(* Logix 5000 project; controller Capstone_PLC_1 1769-L16ER-BB1B rev 38.11; software revision 38.00 *)

TASK MainTask (continuous, watchdog 500 ms) : MainProgram, SecondaryProgram

MODULES
   Local : 1769-L16ER-BB1B (PointIO 0, rev 38.11)
      Point_IO : 1734-AENTR (Ethernet 192.168.1.30, rev 4.1, Output RPI 20 ms)   // Extended I/O for PLC
         POINT_DI_1 : 1734-IB8 (PointIO 1, rev 3.1)   // Sensors from tray to color identification
              Point_IO:1:I.2   // Induction sensor 2 - Extended I/O DI (1734-IB8, Slot 1, Channel 2)
              Point_IO:1:I.1   // Induction sensor 1 - Extended I/O DI (1734-IB8, Slot 1, Channel 1)
              Point_IO:1:I.0   // Tray present limit switch - Extended I/O DI (1734-IB8, Slot 1, Channel 0)
              Point_IO:1:I.3   // Induction sensor 3 - Extended I/O DI (1734-IB8, Slot 1, Channel 3)
              Point_IO:1:I.4   // Through beam sensor 1 - Extended I/O DI (1734-IB8, Slot 1, Channel 4)
              Point_IO:1:I.5   // Through beam sensor 2 - Extended I/O DI (1734-IB8, Slot 1, Channel 5)
         POINT_DI_2 : 1734-IB8 (PointIO 2, rev 3.1)   // Sorting sensors
              Point_IO:2:I.0   // Diffuse sensor, cube on conveyor - Extended I/O DI (1734-IB8, Slot 2, Channel 0)
              Point_IO:2:I.1   // Diffuse sensor, cube at bin 1 - Extended I/O DI (1734-IB8, Slot 2, Channel 1)
              Point_IO:2:I.2   // Diffuse sensor, cube at bin 2 - Extended I/O DI (1734-IB8, Slot 2, Channel 2)
              Point_IO:2:I.3   // Diffuse sensor, cube at bin 3 - Extended I/O DI (1734-IB8, Slot 2, Channel 3)
              Point_IO:2:I.4   // Diffuse sensor, cube at reject bin - Extended I/O DI (1734-IB8, Slot 2, Channel 4)
              Point_IO:2:I.5   // Input for color sensor bit 0
              Point_IO:2:I.6   // Input for color sensor bit 1
              Point_IO:2:I.7   // Input for color sensor bit 2
         POINT_DO_3 : 1734-OB8E (PointIO 3, rev 3.1)   // Conveyor, eject nozzles
              Point_IO:3:O.0   // Output for conveyor - Extended I/O DO (1734-OB8E, Slot 3, Channel 0)
              Point_IO:3:O.1   // Output for eject nozzle 1- Extended I/O DO (1734-OB8E, Slot 3, Channel 1)
              Point_IO:3:O.2   // Output for eject nozzle 2- Extended I/O DO (1734-OB8E, Slot 3, Channel 2)
              Point_IO:3:O.3   // Output for eject nozzle 3- Extended I/O DO (1734-OB8E, Slot 3, Channel 3)
      Discrete_IO : Embedded (PointIO 1, rev 38.1, Output RPI 20 ms)
END_MODULES

VAR_GLOBAL   (* controller tags *)
   At_Destination : BOOL;   // Tracks if the sorted cube has reached the correct bin
   Cmd_Conv : ALIAS FOR Point_IO:3:O.0;   // Logically commands conveyor output
   Cmd_Eject_1 : ALIAS FOR Point_IO:3:O.1;   // Logically commands ejection nozzle 1 output
   Cmd_Eject_2 : ALIAS FOR Point_IO:3:O.2;   // Logically commands ejection nozzle 2 output
   Cmd_Eject_3 : ALIAS FOR Point_IO:3:O.3;   // Logically commands ejection nozzle 3 output
   COL_DET : DINT := 4;   // State, detecting color
   Color_Bit_0 : ALIAS FOR Point_IO:2:I.5;   // Input from color sensor configured in Binary Out
   Color_Bit_1 : ALIAS FOR Point_IO:2:I.6;   // Input from color sensor configured in Binary Out
   Color_Bit_2 : ALIAS FOR Point_IO:2:I.7;   // Input from color sensor configured in Binary Out
   Color_Captured : BOOL;   // Triggers when a color has been identified successfully
   Color_Code : DINT;   // Detected color code
   ColorValid : BOOL;   // Validates color reading
   Con_0 : DINT;   // Constant 0
   Con_1 : DINT := 1;   // Constant 1
   Con_2 : DINT := 2;   // Constant 2
   Con_3 : DINT := 3;   // Constant 3
   Con_4 : DINT := 4;   // Constant 4
   Conv_Active : BOOL;   // Controls conveyor
   Count_1 : DINT;   // Bin 1 counter
   Count_2 : DINT;   // Bin 2 counter
   Count_3 : DINT;   // Bin 3 counter
   Count_4 : DINT;   // Bin 4 counter
   Dest_Bin : DINT;   // Stores destination bin after a cube is identified
   Destination_Known : BOOL;
   Detected_Color : DINT;   // Stores detected color code
   Dif_Bin_1 : ALIAS FOR Point_IO:2:I.1;   // Diffuse sensor: Bin 1
   Dif_Bin_2 : ALIAS FOR Point_IO:2:I.2;   // Diffuse sensor: Bin 2
   Dif_Bin_3 : ALIAS FOR Point_IO:2:I.3;   // Diffuse sensor: Bin 3
   Dif_Conv : ALIAS FOR Point_IO:2:I.0;   // Part detected on conveyor start position
   DONE : DINT := 7;   // State, cube sorted, triggers check, if cubes left to be sorted State returns to PICK, if not State returns to IDLE
   E_Stop : BOOL;   // Emergency stop, disables all outputs
   Eject_1 : BOOL;   // Controls ejection nozzle at bin 1
   Eject_2 : BOOL;   // Controls ejection nozzle at bin 2
   Eject_3 : BOOL;   // Controls ejection nozzle at bin 3
   FAULT : DINT := 99;
   HMI_Init_Sys : BOOL;   // HMI Input: Triggers SPEL_Init
   HMI_PB1 : ALIAS FOR STOP;   // HMI RED PB
   HMI_PB2 : BOOL;   // HMI ORANGE PB
   HMI_PB3 : ALIAS FOR START;   // HMI GREEN PB
   HMI_PB4 : BOOL;   // HMI BLUE PB
   HMI_Reset : BOOL;   // HMI Input to reset sysm to idle state
   IDLE : DINT := 1;   // State, system is initialized but no tray is present or tray present with no cubes
   Ind_Tray_1 : ALIAS FOR Point_IO:1:I.1;   // Induction sensor 1: Tray identification
   Ind_Tray_2 : ALIAS FOR Point_IO:1:I.2;   // Induction sensor 2: Tray identification
   Ind_Tray_3 : ALIAS FOR Point_IO:1:I.3;   // Induction sensor 3: Tray identification
   INIT : DINT;   // State, waiting for initialization conditions
   Lim_Tray_Pres : ALIAS FOR Point_IO:1:I.0;   // Limit switch: Tray presence
   OS_Col_Det : BOOL;   // Ensures color detetion only happens once on subroutine entry
   OS_Col_Det_State : BOOL;   // One shot ensures Col_Det state triggers cleanly
   OS_ColorValid : BOOL;   // Prevents multiple color readings at the same time
   OS_Conv : BOOL;   // One shot ensure clean transition to conveyor state
   OS_Init : BOOL;   // One shot keeps init executing once
   OS_Ready : BOOL;   // One shot protects IDLE > READY state transition
   OS_Reset : BOOL;   // One shot for reset to prevent it from triggering multiple times on a single press
   OS_Sort : BOOL;   // One shot ensure clean transition to sort state
   OS_Sort_Done : BOOL;   // One shot ensure clean entry into done state
   OS_Start : BOOL;   // One shot protects start production from triggering multiple times on input
   OS_TrayID_1 : BOOL;   // Protects from induction sensor reading multipletimes
   OS_TrayID_2 : BOOL;   // Protects from induction sensor reading multipletimes
   OS_TrayID_3 : BOOL;   // Protects from induction sensor reading multipletimes
   Output_Enable : BOOL;   // Enables outputs if robot initialized, system in run mode, and no faults or estop
   PB1 : ALIAS FOR Local:1:I.Data.0;   // RED PB
   PB2 : ALIAS FOR Local:1:I.Data.1;   // ORANGE PB
   PB3 : ALIAS FOR Local:1:I.Data.2;   // GREEN PB
   PB4 : ALIAS FOR Local:1:I.Data.3;   // BLUE PB
   PICK : DINT := 3;   // State, robot picking
   Pick_Done : BOOL;   // Triggers when SPEL pick is completed
   Pick_Index : DINT;   // Tracks cubes on tray for picking
   PL1 : ALIAS FOR Local:1:O.Data.0;   // RED LIGHT
   PL2 : ALIAS FOR Local:1:O.Data.1;   // ORANGE LIGHT
   PL3 : ALIAS FOR Local:1:O.Data.2;   // GREEN LIGHT
   PL4 : ALIAS FOR Local:1:O.Data.3;   // BLUE LIGHT
   PLACE_AOI : BOOL;
   Place_Done : BOOL;
   READY : DINT := 2;   // State, Tray and cubes present
   Rec_Color_Bin_1 : DINT;   // HMI input: color assigned to bin 1
   Rec_Color_Bin_2 : DINT;   // HMI input: color assigned to bin 2
   Rec_Color_Bin_3 : DINT;   // HMI input: color assigned to bin 3
   Rec_Color_Bin_4 : DINT;   // HMI input: color assigned to bin 4 "reject"
   ROBOT_BUSY : BOOL;
   ROBOT_DONE : BOOL;
   ROBOT_INIT : BOOL;
   Robot_Initialized : BOOL;   // Checks if robot is ready for production
   ROBOT_PICK_1 : BOOL;
   ROBOT_PICK_2 : BOOL;
   ROBOT_PICK_3 : BOOL;
   ROBOT_PICK_4 : BOOL;
   ROBOT_READY : BOOL;
   SCADA_Color : DINT;   // SCADA tag shows identified color
   SCADA_Conv : BOOL;   // SCADA tag shows conveyor activity
   SCADA_Count_1 : DINT;   // SCADA tag shows counter for bin 1
   SCADA_Count_2 : DINT;   // SCADA tag shows counter for bin 2
   SCADA_Count_3 : DINT;   // SCADA tag shows counter for bin 3
   SCADA_Count_4 : DINT;   // SCADA tag shows counter for bin 4
   SCADA_Dest : DINT;   // SCADA tag shows destination bin
   SCADA_State : DINT;   // SCADA tag shows current system state
   SCADA_TrayID : DINT;   // SCADA tag shows Tray ID
   SORT : DINT := 6;   // State, cube on conveyor
   Sort_Done : BOOL;   // Tracks if sorting is done
   SPEL_Init : BOOL;   // Triggers SPEL_Init AOI
   SPEL_Init_Done : BOOL;   // Checks if SPEL_Init is completed
   START : BOOL;   // Start production, triggered by PB3 (green) or HMI input
   State : DINT;   // Tracks system state for control flow
   STOP : BOOL;   // Stops production, triggered by PB1 (red) or HMI input
   Sys_Fault : BOOL;   // Enabled for any fault condition
   Sys_Rdy : BOOL;   // System staged and safe for production
   Sys_Run : BOOL;   // Production active
   TEST_Color_Entry : BOOL;   // User controlled bit for entering color detation, used for testing/debugging
   Thr_Cubes_1 : ALIAS FOR Point_IO:1:I.4;   // Through beam sensor: identifies cube presence in tray row 1
   Thr_Cubes_2 : ALIAS FOR Point_IO:1:I.5;   // Through beam sensor: identifies cube presence in tray row 2
   TIMER_BLINK_1 : TIMER := (PRE := 500);
   TIMER_BLINK_2 : TIMER := (PRE := 500);
   TIMER_EJECT_1 : TIMER := (PRE := 200);
   TIMER_EJECT_2 : TIMER := (PRE := 200);
   TIMER_EJECT_3 : TIMER := (PRE := 200);
   TIMER_REJECT : TIMER := (PRE := 8000);
   TMR_Color_Read : TIMER := (PRE := 500);   // Delays color sensor input for validation
   TO_CONV : DINT := 5;   // State, moving cube to conveyor
   Tray_Full : BOOL;   // Energizes if both through beam sensors are triggered for cube presence
   TrayID : DINT;   // Calculated tray ID from induction sensors
   TrayIdentified : BOOL;   // Tracks if a tray is identified
END_VAR

PROGRAM MainProgram   (* main routine MainRoutine *)

ROUTINE Blinker_Fault   (* ladder *)
// Flashes red light to indicate system fault
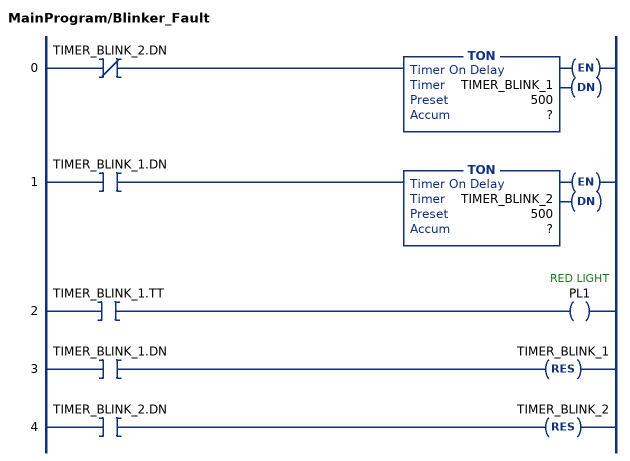
   0: XIO(TIMER_BLINK_2.DN)TON(TIMER_BLINK_1,?,?);
   1: XIC(TIMER_BLINK_1.DN)TON(TIMER_BLINK_2,?,?);
   2: XIC(TIMER_BLINK_1.TT)OTE(PL1);
   3: XIC(TIMER_BLINK_1.DN)RES(TIMER_BLINK_1);
   4: XIC(TIMER_BLINK_2.DN)RES(TIMER_BLINK_2);
END_ROUTINE

ROUTINE Blinker_Init   (* ladder *)
// Flashes blue light to show system ready for initialization
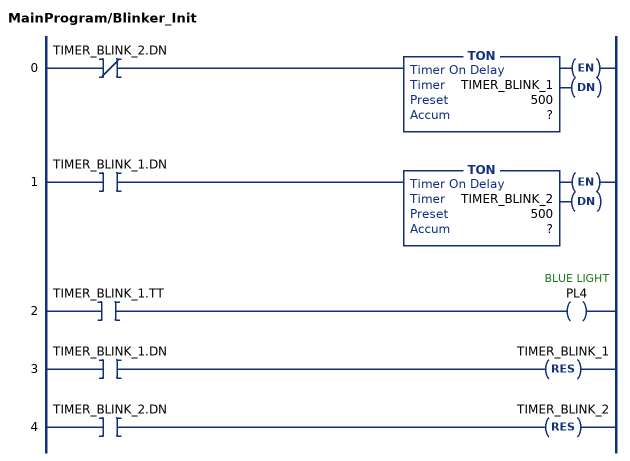
   0: XIO(TIMER_BLINK_2.DN)TON(TIMER_BLINK_1,?,?);
   1: XIC(TIMER_BLINK_1.DN)TON(TIMER_BLINK_2,?,?);
   2: XIC(TIMER_BLINK_1.TT)OTE(PL4);
   3: XIC(TIMER_BLINK_1.DN)RES(TIMER_BLINK_1);
   4: XIC(TIMER_BLINK_2.DN)RES(TIMER_BLINK_2);
END_ROUTINE

ROUTINE Blinker_Initialized   (* ladder *)
// Flashes green light to show system initialized
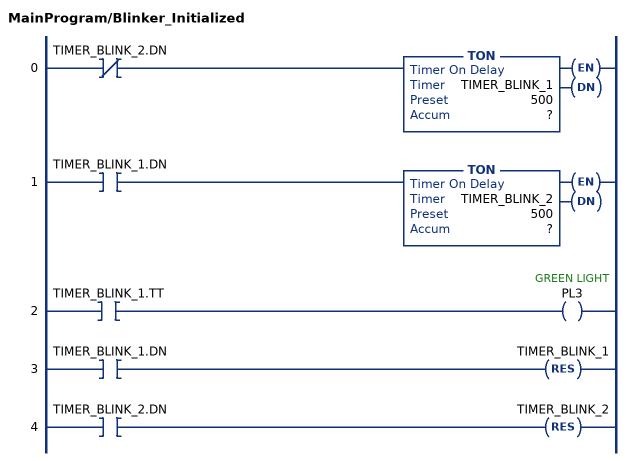
   0: XIO(TIMER_BLINK_2.DN)TON(TIMER_BLINK_1,?,?);
   1: XIC(TIMER_BLINK_1.DN)TON(TIMER_BLINK_2,?,?);
   2: XIC(TIMER_BLINK_1.TT)OTE(PL3);
   3: XIC(TIMER_BLINK_1.DN)RES(TIMER_BLINK_1);
   4: XIC(TIMER_BLINK_2.DN)RES(TIMER_BLINK_2);
END_ROUTINE

ROUTINE Blinker_Running   (* ladder *)
// Flashes orange light to show system running
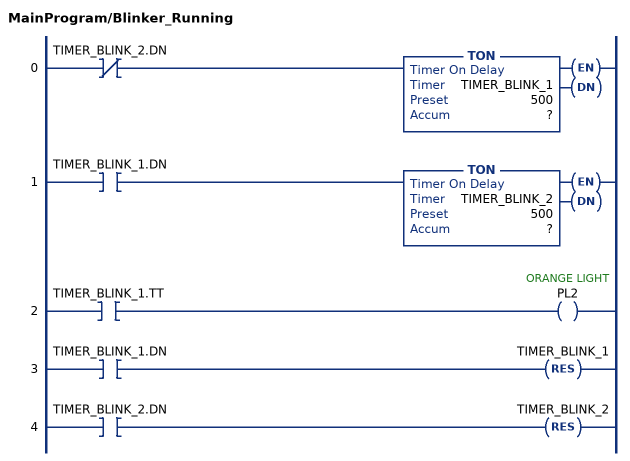
   0: XIO(TIMER_BLINK_2.DN)TON(TIMER_BLINK_1,?,?);
   1: XIC(TIMER_BLINK_1.DN)TON(TIMER_BLINK_2,?,?);
   2: XIC(TIMER_BLINK_1.TT)OTE(PL2);
   3: XIC(TIMER_BLINK_1.DN)RES(TIMER_BLINK_1);
   4: XIC(TIMER_BLINK_2.DN)RES(TIMER_BLINK_2);
END_ROUTINE

ROUTINE Color_Detect   (* ladder *)
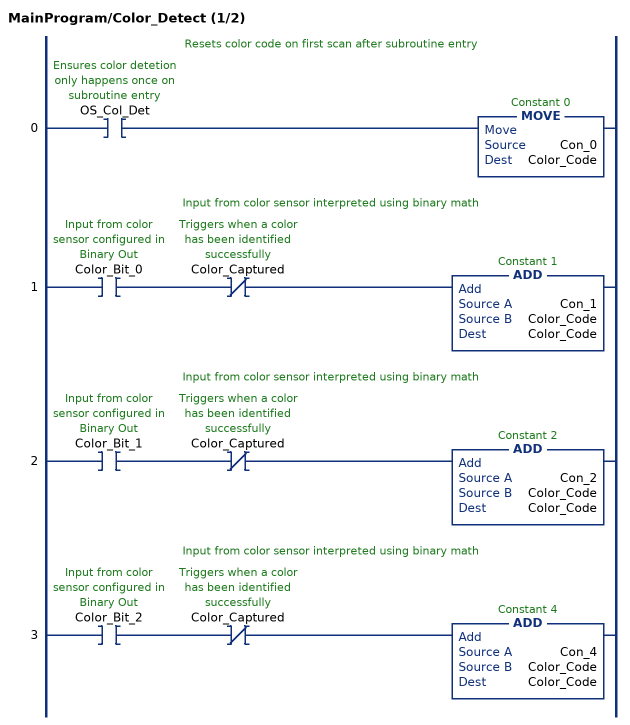
   // Resets color code on first scan after subroutine entry
   0: XIC(OS_Col_Det)MOVE(Con_0,Color_Code);
   // Input from color sensor interpreted using binary math
   1: XIC(Color_Bit_0)XIO(Color_Captured)ADD(Con_1,Color_Code,Color_Code);
   // Input from color sensor interpreted using binary math
   2: XIC(Color_Bit_1)XIO(Color_Captured)ADD(Con_2,Color_Code,Color_Code);
   // Input from color sensor interpreted using binary math
   3: XIC(Color_Bit_2)XIO(Color_Captured)ADD(Con_4,Color_Code,Color_Code);
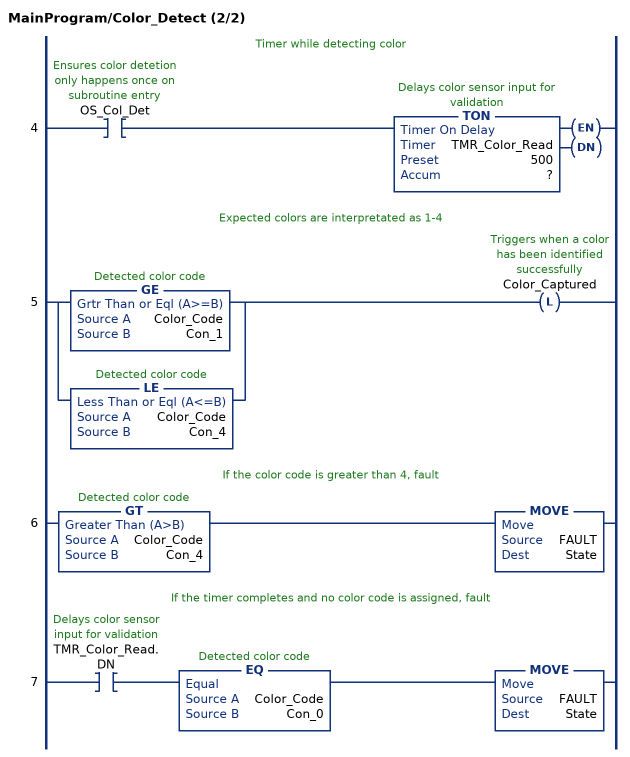
   // Timer while detecting color
   4: XIC(OS_Col_Det)TON(TMR_Color_Read,?,?);
   // Expected colors are interpretated as 1-4
   5: [GE(Color_Code,Con_1) ,LE(Color_Code,Con_4) ]OTL(Color_Captured);
   // If the color code is greater than 4, fault
   6: GT(Color_Code,Con_4)MOVE(FAULT,State);
   // If the timer completes and no color code is assigned, fault
   7: XIC(TMR_Color_Read.DN)EQ(Color_Code,Con_0)MOVE(FAULT,State);
END_ROUTINE

ROUTINE Control_Done   (* ladder *)
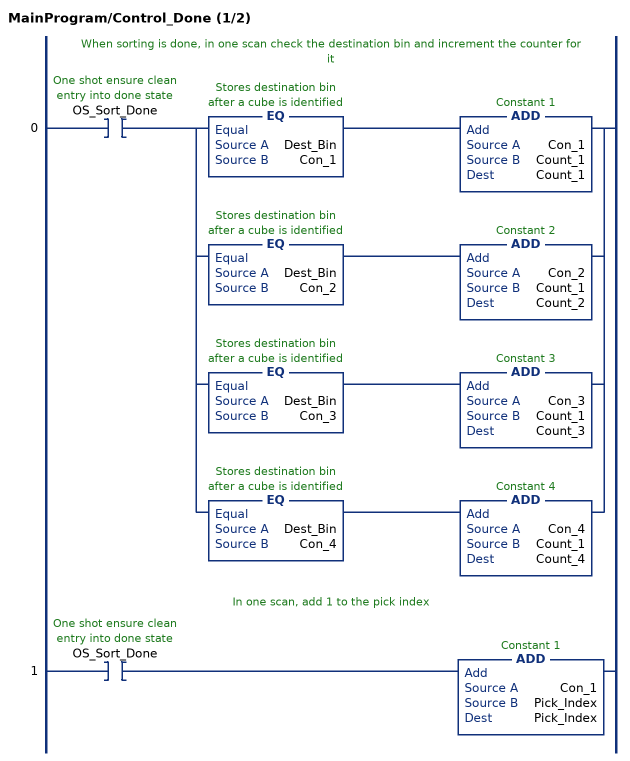
   // When sorting is done, in one scan check the destination bin and increment the counter for it
   0: XIC(OS_Sort_Done)[EQ(Dest_Bin,Con_1) ADD(Con_1,Count_1,Count_1) ,[EQ(Dest_Bin,Con_2) ADD(Con_2,Count_1,Count_2) ,[EQ(Dest_Bin,Con_3) ADD(Con_3,Count_1,Count_3) ,EQ(Dest_Bin,Con_4) ADD(Con_4,Count_1,Count_4) ] ] ];
   // In one scan, add 1 to the pick index
   1: XIC(OS_Sort_Done)ADD(Con_1,Pick_Index,Pick_Index);
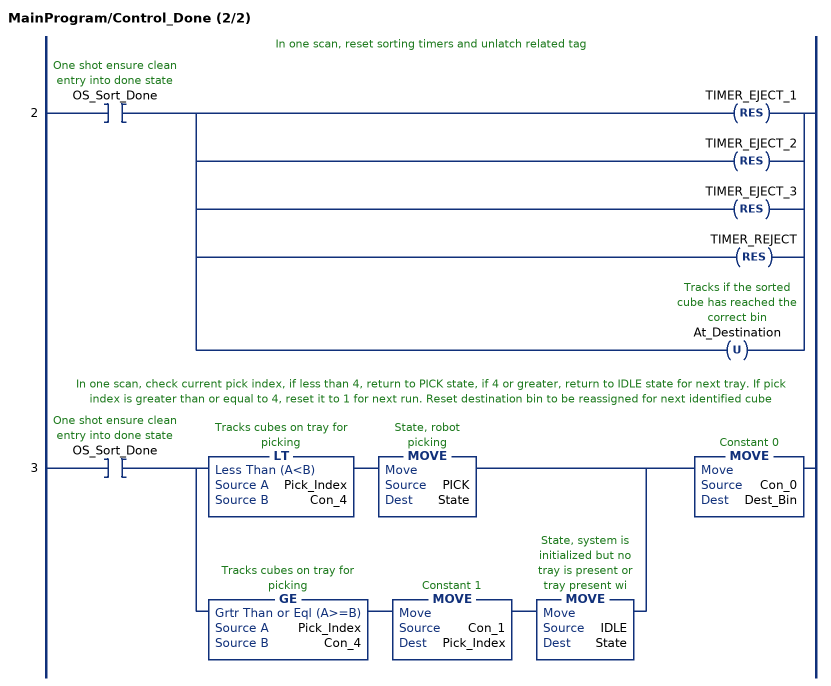
   // In one scan, reset sorting timers and unlatch related tag
   2: XIC(OS_Sort_Done)[RES(TIMER_EJECT_1) ,[RES(TIMER_EJECT_2) ,[RES(TIMER_EJECT_3) ,[RES(TIMER_REJECT) ,OTU(At_Destination) ] ] ] ];
   // In one scan, check current pick index, if less than 4, return to PICK state, if 4 or greater, return to IDLE state for next tray. If pick index is greater than or equal to 4, reset it to 1 for next run. Reset destination bin to be reassigned for next identified cube
   3: XIC(OS_Sort_Done)[LT(Pick_Index,Con_4) MOVE(PICK,State) ,GE(Pick_Index,Con_4) MOVE(Con_1,Pick_Index) MOVE(IDLE,State) ]MOVE(Con_0,Dest_Bin);
END_ROUTINE

ROUTINE Control_Lights   (* ladder *)
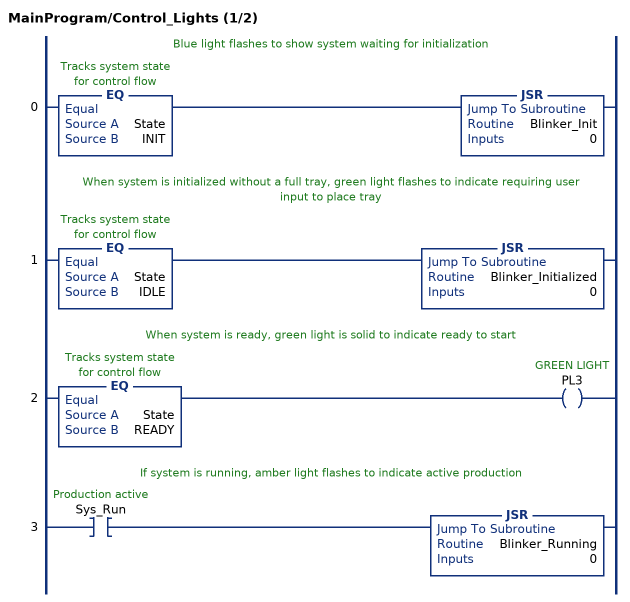
   // Blue light flashes to show system waiting for initialization
   0: EQ(State,INIT)JSR(Blinker_Init,0);
   // When system is initialized without a full tray, green light flashes to indicate requiring user input to place tray
   1: EQ(State,IDLE)JSR(Blinker_Initialized,0);
   // When system is ready, green light is solid to indicate ready to start
   2: EQ(State,READY)OTE(PL3);
   // If system is running, amber light flashes to indicate active production
   3: XIC(Sys_Run)JSR(Blinker_Running,0);
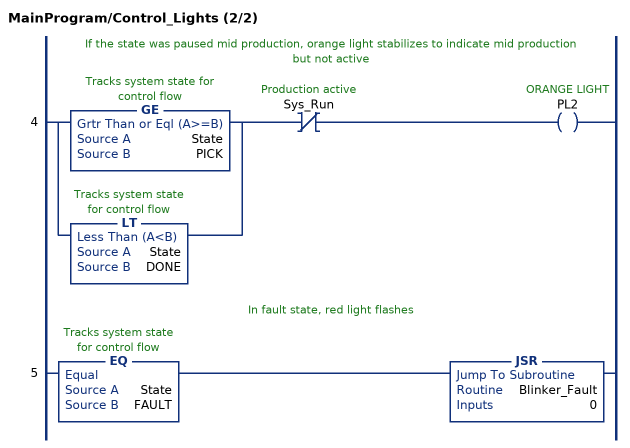
   // If the state was paused mid production, orange light stabilizes to indicate mid production but not active
   4: [GE(State,PICK) ,LT(State,DONE) ]XIO(Sys_Run)OTE(PL2);
   // In fault state, red light flashes
   5: EQ(State,FAULT)JSR(Blinker_Fault,0);
END_ROUTINE

ROUTINE Control_Pick   (* ladder *)
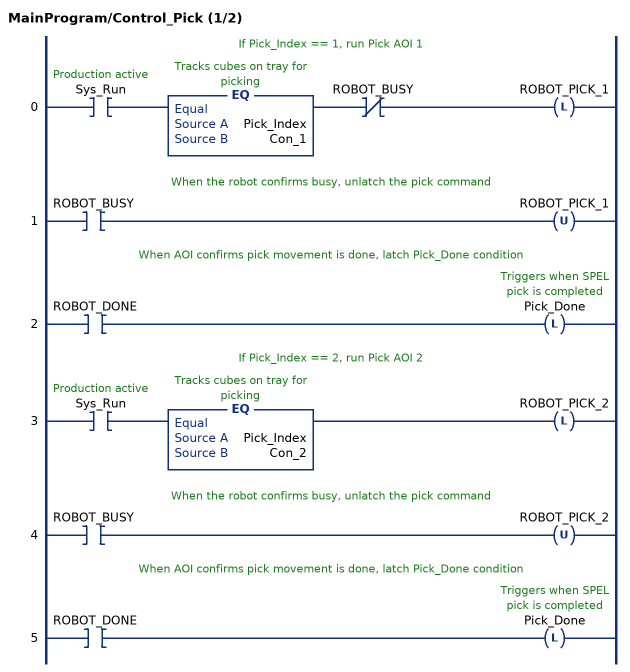
   // If Pick_Index == 1, run Pick AOI 1
   0: XIC(Sys_Run)EQ(Pick_Index,Con_1)XIO(ROBOT_BUSY)OTL(ROBOT_PICK_1);
   // When the robot confirms busy, unlatch the pick command
   1: XIC(ROBOT_BUSY)OTU(ROBOT_PICK_1);
   // When AOI confirms pick movement is done, latch Pick_Done condition
   2: XIC(ROBOT_DONE)OTL(Pick_Done);
   // If Pick_Index == 2, run Pick AOI 2
   3: XIC(Sys_Run)EQ(Pick_Index,Con_2)OTL(ROBOT_PICK_2);
   // When the robot confirms busy, unlatch the pick command
   4: XIC(ROBOT_BUSY)OTU(ROBOT_PICK_2);
   // When AOI confirms pick movement is done, latch Pick_Done condition
   5: XIC(ROBOT_DONE)OTL(Pick_Done);
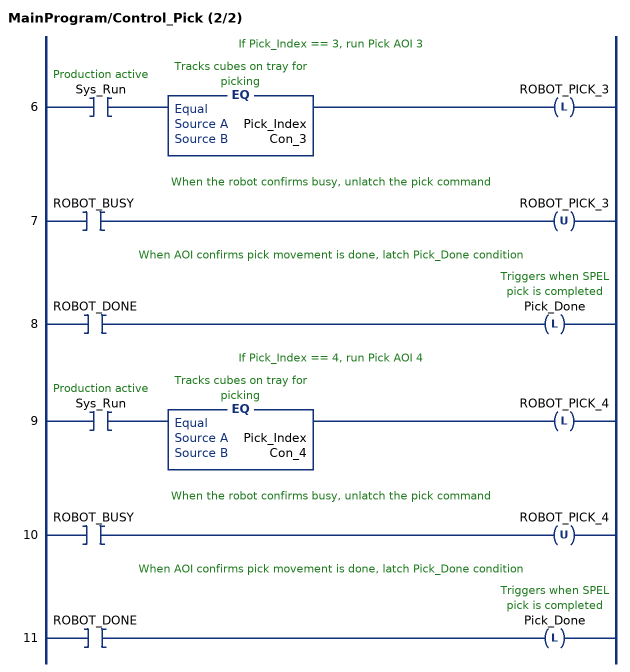
   // If Pick_Index == 3, run Pick AOI 3
   6: XIC(Sys_Run)EQ(Pick_Index,Con_3)OTL(ROBOT_PICK_3);
   // When the robot confirms busy, unlatch the pick command
   7: XIC(ROBOT_BUSY)OTU(ROBOT_PICK_3);
   // When AOI confirms pick movement is done, latch Pick_Done condition
   8: XIC(ROBOT_DONE)OTL(Pick_Done);
   // If Pick_Index == 4, run Pick AOI 4
   9: XIC(Sys_Run)EQ(Pick_Index,Con_4)OTL(ROBOT_PICK_4);
   // When the robot confirms busy, unlatch the pick command
   10: XIC(ROBOT_BUSY)OTU(ROBOT_PICK_4);
   // When AOI confirms pick movement is done, latch Pick_Done condition
   11: XIC(ROBOT_DONE)OTL(Pick_Done);
END_ROUTINE

ROUTINE Control_Sort   (* ladder *)
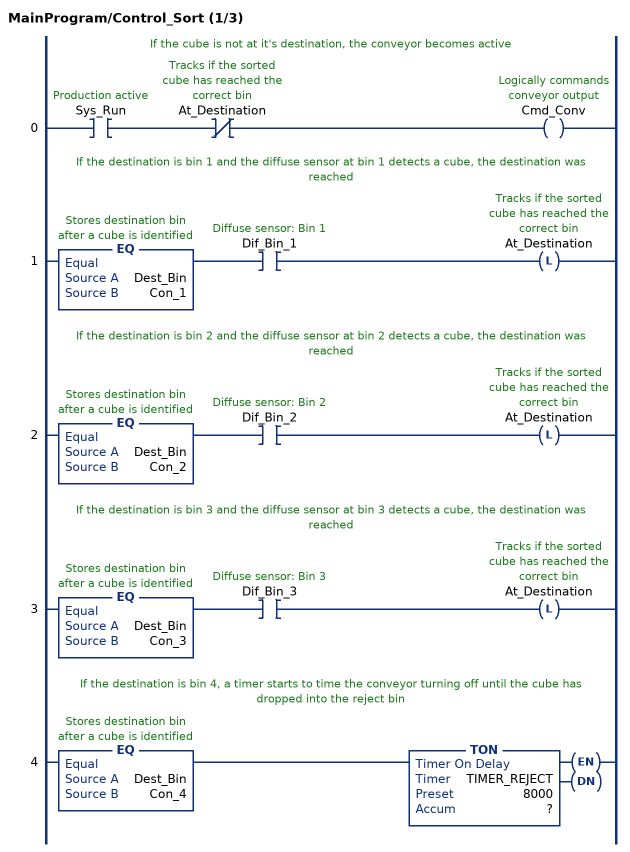
   // If the cube is not at it's destination, the conveyor becomes active
   0: XIC(Sys_Run)XIO(At_Destination)OTE(Cmd_Conv);
   // If the destination is bin 1 and the diffuse sensor at bin 1 detects a cube, the destination was reached
   1: EQ(Dest_Bin,Con_1)XIC(Dif_Bin_1)OTL(At_Destination);
   // If the destination is bin 2 and the diffuse sensor at bin 2 detects a cube, the destination was reached
   2: EQ(Dest_Bin,Con_2)XIC(Dif_Bin_2)OTL(At_Destination);
   // If the destination is bin 3 and the diffuse sensor at bin 3 detects a cube, the destination was reached
   3: EQ(Dest_Bin,Con_3)XIC(Dif_Bin_3)OTL(At_Destination);
   // If the destination is bin 4, a timer starts to time the conveyor turning off until the cube has dropped into the reject bin
   4: EQ(Dest_Bin,Con_4)TON(TIMER_REJECT,?,?);
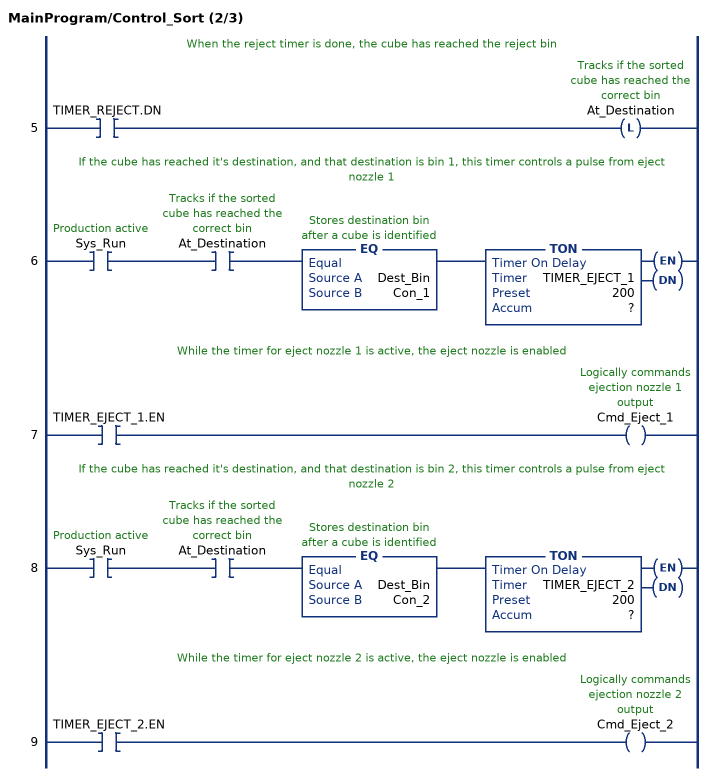
   // When the reject timer is done, the cube has reached the reject bin
   5: XIC(TIMER_REJECT.DN)OTL(At_Destination);
   // If the cube has reached it's destination, and that destination is bin 1, this timer controls a pulse from eject nozzle 1
   6: XIC(Sys_Run)XIC(At_Destination)EQ(Dest_Bin,Con_1)TON(TIMER_EJECT_1,?,?);
   // While the timer for eject nozzle 1 is active, the eject nozzle is enabled
   7: XIC(TIMER_EJECT_1.EN)OTE(Cmd_Eject_1);
   // If the cube has reached it's destination, and that destination is bin 2, this timer controls a pulse from eject nozzle 2
   8: XIC(Sys_Run)XIC(At_Destination)EQ(Dest_Bin,Con_2)TON(TIMER_EJECT_2,?,?);
   // While the timer for eject nozzle 2 is active, the eject nozzle is enabled
   9: XIC(TIMER_EJECT_2.EN)OTE(Cmd_Eject_2);
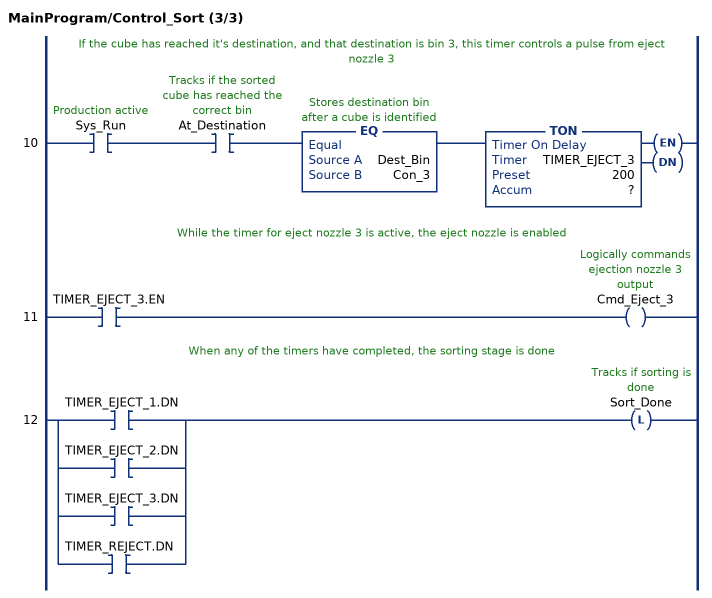
   // If the cube has reached it's destination, and that destination is bin 3, this timer controls a pulse from eject nozzle 3
   10: XIC(Sys_Run)XIC(At_Destination)EQ(Dest_Bin,Con_3)TON(TIMER_EJECT_3,?,?);
   // While the timer for eject nozzle 3 is active, the eject nozzle is enabled
   11: XIC(TIMER_EJECT_3.EN)OTE(Cmd_Eject_3);
   // When any of the timers have completed, the sorting stage is done
   12: [XIC(TIMER_EJECT_1.DN) ,[XIC(TIMER_EJECT_2.DN) ,[XIC(TIMER_EJECT_3.DN) ,XIC(TIMER_REJECT.DN) ] ] ]OTL(Sort_Done);
END_ROUTINE

ROUTINE Control_To_Conveyor   (* ladder *)
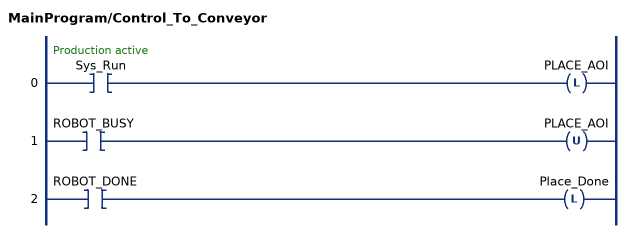
   0: XIC(Sys_Run)OTL(PLACE_AOI);
   1: XIC(ROBOT_BUSY)OTU(PLACE_AOI);
   2: XIC(ROBOT_DONE)OTL(Place_Done);
END_ROUTINE

ROUTINE Determine_Destination   (* ladder *)
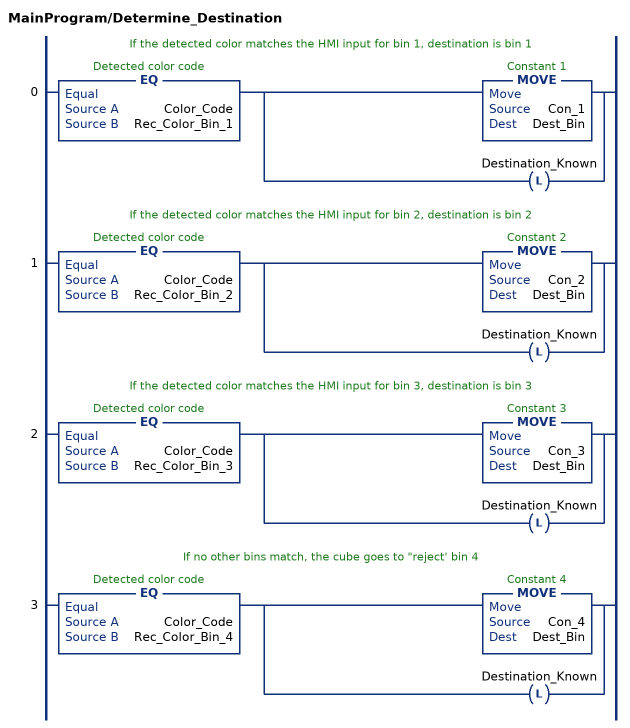
   // If the detected color matches the HMI input for bin 1, destination is bin 1
   0: EQ(Color_Code,Rec_Color_Bin_1)[MOVE(Con_1,Dest_Bin) ,OTL(Destination_Known) ];
   // If the detected color matches the HMI input for bin 2, destination is bin 2
   1: EQ(Color_Code,Rec_Color_Bin_2)[MOVE(Con_2,Dest_Bin) ,OTL(Destination_Known) ];
   // If the detected color matches the HMI input for bin 3, destination is bin 3
   2: EQ(Color_Code,Rec_Color_Bin_3)[MOVE(Con_3,Dest_Bin) ,OTL(Destination_Known) ];
   // If no other bins match, the cube goes to "reject' bin 4
   3: EQ(Color_Code,Rec_Color_Bin_4)[MOVE(Con_4,Dest_Bin) ,OTL(Destination_Known) ];
END_ROUTINE

ROUTINE MainRoutine   (* ladder *)
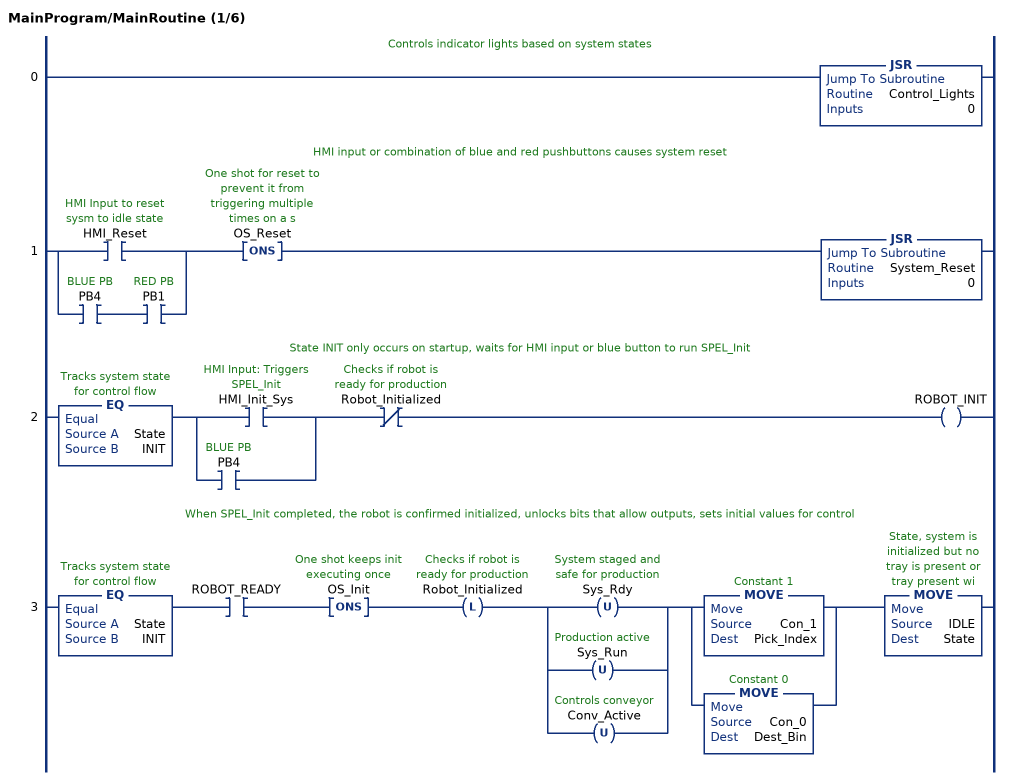
   // Controls indicator lights based on system states
   0: JSR(Control_Lights,0);
   // HMI input or combination of blue and red pushbuttons causes system reset
   1: [XIC(HMI_Reset) ,XIC(PB4) XIC(PB1) ]ONS(OS_Reset)JSR(System_Reset,0);
   // State INIT only occurs on startup, waits for HMI input or blue button to run SPEL_Init
   2: EQ(State,INIT)[XIC(HMI_Init_Sys) ,XIC(PB4) ]XIO(Robot_Initialized)OTE(ROBOT_INIT);
   // When SPEL_Init completed, the robot is confirmed initialized, unlocks bits that allow outputs, sets initial values for control
   3: EQ(State,INIT)XIC(ROBOT_READY)ONS(OS_Init)OTL(Robot_Initialized)[OTU(Sys_Rdy) ,[OTU(Sys_Run) ,OTU(Conv_Active) ] ][MOVE(Con_1,Pick_Index) ,MOVE(Con_0,Dest_Bin) ]MOVE(IDLE,State);
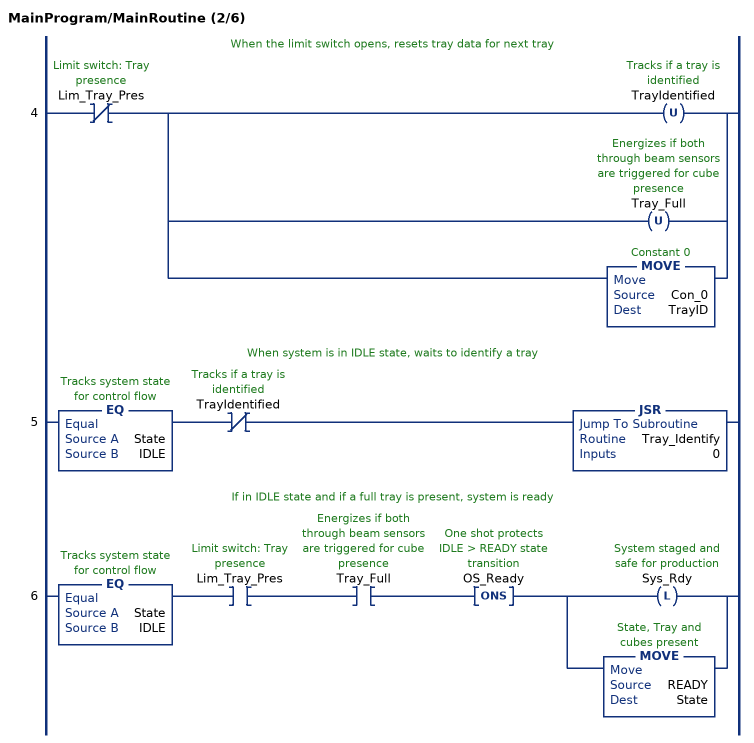
   // When the limit switch opens, resets tray data for next tray
   4: XIO(Lim_Tray_Pres)[OTU(TrayIdentified) ,[OTU(Tray_Full) ,MOVE(Con_0,TrayID) ] ];
   // When system is in IDLE state, waits to identify a tray
   5: EQ(State,IDLE)XIO(TrayIdentified)JSR(Tray_Identify,0);
   // If in IDLE state and if a full tray is present, system is ready
   6: EQ(State,IDLE)XIC(Lim_Tray_Pres)XIC(Tray_Full)ONS(OS_Ready)[OTL(Sys_Rdy) ,MOVE(READY,State) ];
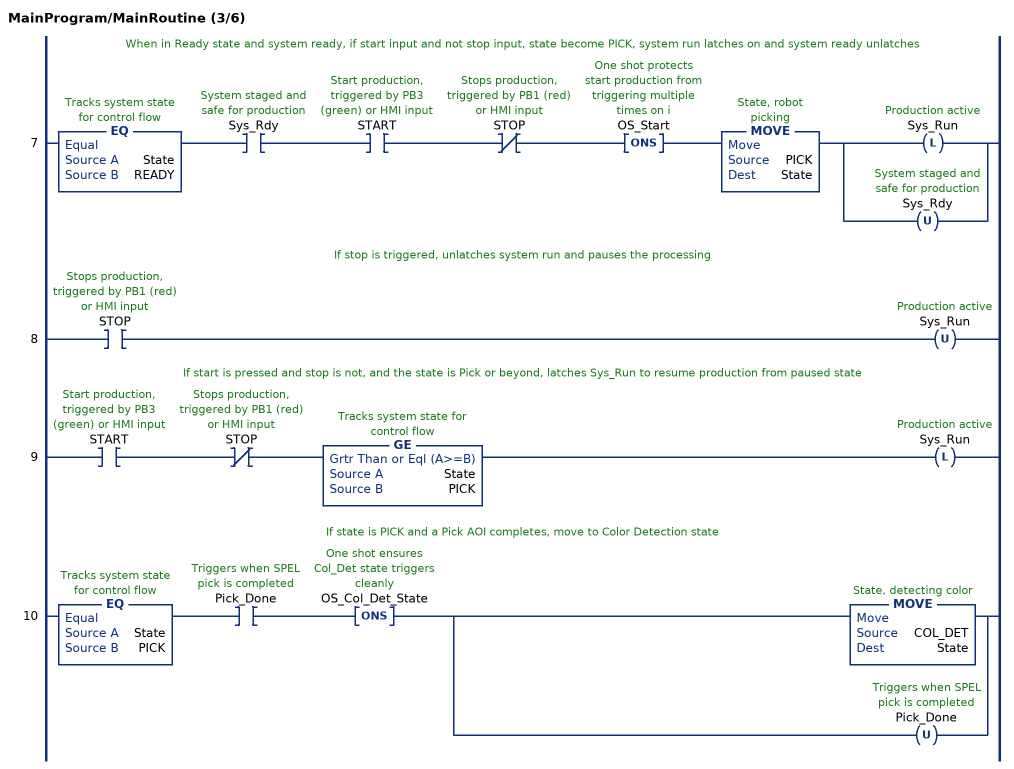
   // When in Ready state and system ready, if start input and not stop input, state become PICK, system run latches on and system ready unlatches
   7: EQ(State,READY)XIC(Sys_Rdy)XIC(START)XIO(STOP)ONS(OS_Start)MOVE(PICK,State)[OTL(Sys_Run) ,OTU(Sys_Rdy) ];
   // If stop is triggered, unlatches system run and pauses the processing
   8: XIC(STOP)OTU(Sys_Run);
   // If start is pressed and stop is not, and the state is Pick or beyond, latches Sys_Run to resume production from paused state
   9: XIC(START)XIO(STOP)GE(State,PICK)OTL(Sys_Run);
   // If state is PICK and a Pick AOI completes, move to Color Detection state
   10: EQ(State,PICK)XIC(Pick_Done)ONS(OS_Col_Det_State)[MOVE(COL_DET,State) ,OTU(Pick_Done) ];
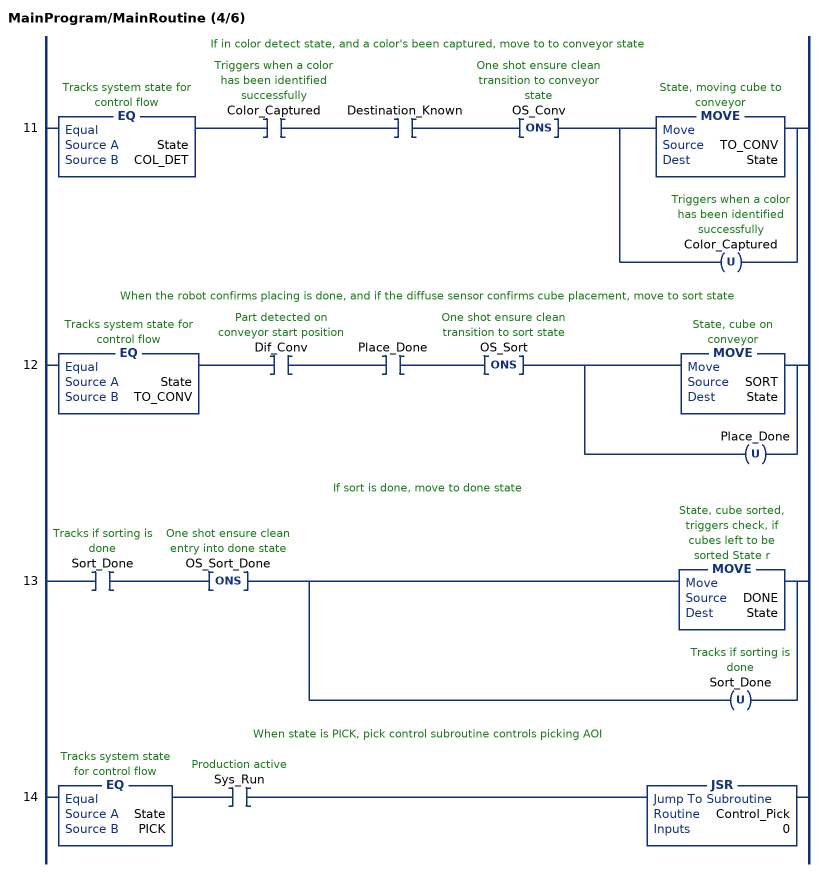
   // If in color detect state, and a color's been captured, move to to conveyor state
   11: EQ(State,COL_DET)XIC(Color_Captured)XIC(Destination_Known)ONS(OS_Conv)[MOVE(TO_CONV,State) ,OTU(Color_Captured) ];
   // When the robot confirms placing is done, and if the diffuse sensor confirms cube placement, move to sort state
   12: EQ(State,TO_CONV)XIC(Dif_Conv)XIC(Place_Done)ONS(OS_Sort)[MOVE(SORT,State) ,OTU(Place_Done) ];
   // If sort is done, move to done state
   13: XIC(Sort_Done)ONS(OS_Sort_Done)[MOVE(DONE,State) ,OTU(Sort_Done) ];
   // When state is PICK, pick control subroutine controls picking AOI
   14: EQ(State,PICK)XIC(Sys_Run)JSR(Control_Pick,0);
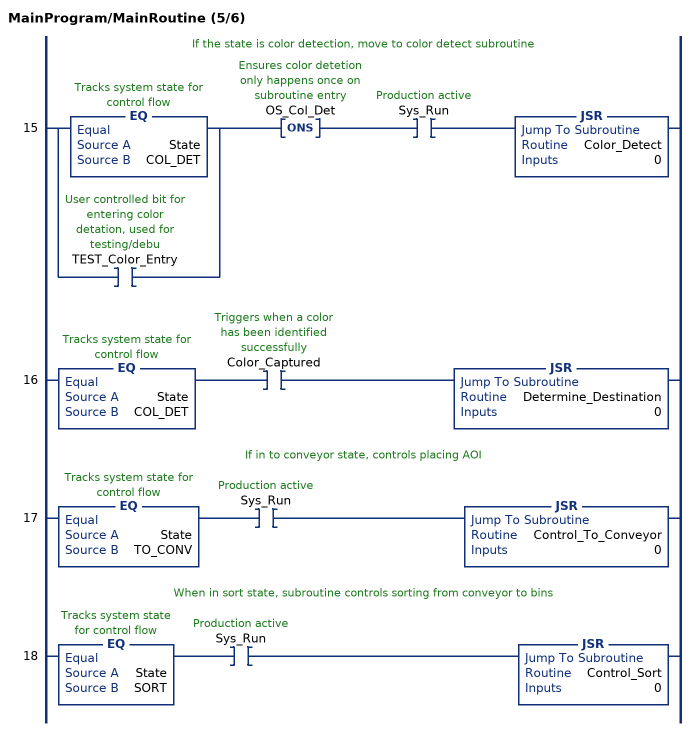
   // If the state is color detection, move to color detect subroutine
   15: [EQ(State,COL_DET) ,XIC(TEST_Color_Entry) ]ONS(OS_Col_Det)XIC(Sys_Run)JSR(Color_Detect,0);
   16: EQ(State,COL_DET)XIC(Color_Captured)JSR(Determine_Destination,0);
   // If in to conveyor state, controls placing AOI
   17: EQ(State,TO_CONV)XIC(Sys_Run)JSR(Control_To_Conveyor,0);
   // When in sort state, subroutine controls sorting from conveyor to bins
   18: EQ(State,SORT)XIC(Sys_Run)JSR(Control_Sort,0);
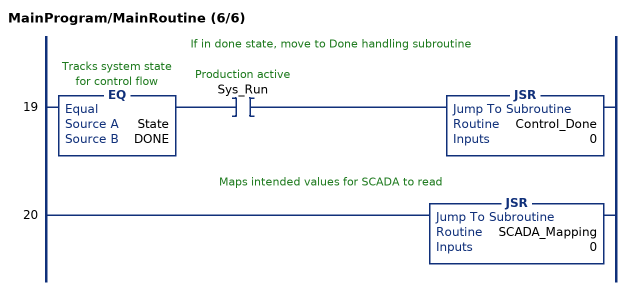
   // If in done state, move to Done handling subroutine
   19: EQ(State,DONE)XIC(Sys_Run)JSR(Control_Done,0);
   // Maps intended values for SCADA to read
   20: JSR(SCADA_Mapping,0);
END_ROUTINE
